FUNCTION_BLOCK FB_Visionsystem EXTENDS GrundstrukturObjekt
VAR_INPUT
END_VAR
VAR_OUTPUT
END_VAR
VAR
END_VAR

END_FUNCTION_BLOCK

(* stored: Version 1.1.0.1
   POU FB_Visionsystem: Id {e5f2d963-b309-4d67-95ab-ab99bcfdaf83}, SpecialFunc None *)
